TYPE ST_GPS_CALCULATIONS :
STRUCT
END_STRUCT
END_TYPE

(* stored: Version 1.1.0.1, ProductVersion 3.1.4022.11
   DUT ST_GPS_CALCULATIONS: Id {8295394f-6ae4-49d8-92af-f6e75391f2c7} *)
